Fanuc KAREL source: kt00418.KL

-- PROVISIONAL review KL for V1013-1; original PC SHA256 e2f2b082760f1543d4cdf6a78322d432c077ee9731e7f9b169fa09e81102c781
-- Incomplete behavior may be omitted. Consult companion uncertainty JSON. Do not deploy.
PROGRAM KT00418
%NOLOCKGROUP
VAR
  OUT : BOOLEAN
-- UNRESOLVED_DECL H1 type=002017
-- UNRESOLVED_DECL H2 type=002017
BEGIN
  -- UNRESOLVED_PC offsets 5-19; opcodes 2E,22,9D,33,B4
  -- UNRESOLVED_PC offsets 24-38; opcodes 2E,22,9D,33,B4
  -- UNRESOLVED_PC offsets 43-57; opcodes 2E,22,9D,33,B4
  -- UNRESOLVED_PC offsets 62-76; opcodes 2E,22,9D,33,B4
  -- UNRESOLVED_PC offsets 81-106; opcodes 22,9D,33,B3,22,9D,33,B3,5B,23
  -- UNRESOLVED_PC offsets 111-115; opcodes 7F
END KT00418
